// TIA Portal V20 export
TYPE "UDT_Service_ParameterDataMedium"
   STRUCT
      used : Array[0..0] of DWord;   // Used configuration parameters of service
      definition : Array[0..31] of "UDT_Service_ParameterDefinition";
   END_STRUCT;
END_TYPE
